// TIA Portal project "Production_Line" (V16)

(* hardware
DEVICE "S7-1200 station_1"  S7-1200 Station
   slot 0: "Rack_0"  S7-1200 Rack  Rack  V1.0
   slot 1: "PLC_1_Storage"  CPU 1214C AC/DC/Rly  6ES7 214-1BG31-0XB0  V3.0
DEVICE "S7-1200 station_2"  S7-1200 Station
   slot 0: "Rack_0"  S7-1200 Rack  Rack  V1.0
   slot 1: "PLC_3_Distribution"  CPU 1214C AC/DC/Rly  6ES7 214-1BG31-0XB0  V3.0
DEVICE "S7-1200 station_3"  S7-1200 Station
   slot 0: "Rack_0"  S7-1200 Rack  Rack  V1.0
   slot 1: "PLC_4_Measuring"  CPU 1214C AC/DC/Rly  6ES7 214-1BG31-0XB0  V3.0
DEVICE "S7-1200 station_4"  S7-1200 Station
   slot 0: "Rack_0"  S7-1200 Rack  Rack  V1.0
   slot 1: "PLC_2_P&P"  CPU 1214C AC/DC/Rly  6ES7 214-1BG31-0XB0  V3.0
DEVICE "S7-1200 station_5"  S7-1200 Station
   slot 0: "Rack_0"  S7-1200 Rack  Rack  V1.0
   slot 1: "PLC_5_Sorting"  CPU 1214C AC/DC/Rly  6ES7 214-1BG31-0XB0  V3.0
DEVICE "HMI4_Measuring"  KTP600 Basic color PN
   slot 0: "HMI4_Measuring"  KTP600 Basic color PN  6AV6 647-0AD11-3AX0  12.0.0.0
   slot 1: "HMI_RT_1"  KTP600 Basic color PN  6AV6 647-0AD11-3AX0  12.0.0.0
   slot 5: "HMI4_Measuring.IE_CP_1"  PROFINET Interface  12.0.0.0
      slot 1: "PROFINET Interface_1"  PROFINET Interface
         slot 1: "Port_1"  Port
DEVICE "HMI1_Storage"  KTP600 Basic color PN
   slot 0: "HMI1_Storage"  KTP600 Basic color PN  6AV6 647-0AD11-3AX0  12.0.0.0
   slot 1: "HMI_RT_2"  KTP600 Basic color PN  6AV6 647-0AD11-3AX0  12.0.0.0
   slot 5: "HMI1_Storage.IE_CP_1"  PROFINET Interface  12.0.0.0
      slot 1: "PROFINET Interface_1"  PROFINET Interface
         slot 1: "Port_1"  Port
*)

// ===== PLC "PLC_1_Storage"  CPU 1214C AC/DC/Rly =====

VAR_GLOBAL   // PLC tag table "Default tag table"
   "Station_homed" AT %I0.0 : Bool;
   "Error" AT %I0.1 : Bool;
   "Busy" AT %I0.2 : Bool;
   "Full" AT %I0.3 : Bool;
   "wp_at_pick" AT %I0.5 : Bool;
   "wp_not_black" AT %I0.6 : Bool;
   "wp_metallic" AT %I0.7 : Bool;
   "Home_station" AT %Q0.0 : Bool;
   "Reset_error" AT %Q0.1 : Bool;
   "Mode" AT %Q0.2 : Bool;
   "bit_0" AT %Q0.3 : Bool;
   "bit_1" AT %Q0.4 : Bool;
   "bit_2" AT %Q0.5 : Bool;
   "Strobe" AT %Q0.6 : Bool;
   "wildcard" AT %Q0.7 : Bool;
   "Rack" AT %MW1 : Int;
   "Color" AT %MW4 : Int;
   "ok" AT %M6.0 : Bool;
END_VAR

// folder: System blocks/Program resources

DATA_BLOCK "IEC_Timer_0_DB"   // DB1
{ S7_Optimized_Access := 'TRUE' }
AUTHOR : Simatic
FAMILY : IEC
NAME : IEC_TMR
VERSION : 1.0
// stored: InstanceOfName IEC_TIMER
"IEC_TIMER"
BEGIN
END_DATA_BLOCK

// folder: (top level)

FUNCTION "Select_color" : Void   // FC1, SCL
{ S7_Optimized_Access := 'TRUE' }
VERSION : 0.1
   VAR_INPUT
      color : Int;
   END_VAR
   VAR_OUTPUT
      bit0 : Bool;
      bit1 : Bool;
      bit2 : Bool;
   END_VAR
BEGIN
   CASE #color OF
       0:// red
           #bit0 := FALSE;
           #bit1 := FALSE;
           #bit2 := FALSE;
       1:// black
           #bit0 := TRUE;
           #bit1 := FALSE;
           #bit2 := FALSE;

       2:  // metallic
           #bit0 := FALSE;
           #bit1 := TRUE;
           #bit2 := FALSE;
       ELSE  // error
           #bit0 := FALSE;
           #bit1 := FALSE;
           #bit2 := FALSE;
   END_CASE;
END_FUNCTION

FUNCTION "Select_rack" : Void   // FC2, SCL
{ S7_Optimized_Access := 'TRUE' }
VERSION : 0.1
   VAR_INPUT
      Rack : Int;
   END_VAR
   VAR_OUTPUT
      bit0 : Bool;
      bit1 : Bool;
      bit2 : Bool;
   END_VAR
BEGIN
   CASE #Rack OF

       1:
           #bit0 := FALSE;
           #bit1 := FALSE;
           #bit2 := FALSE;

       2:
           #bit0 := TRUE;
           #bit1 := FALSE;
           #bit2 := FALSE;
       3:
           #bit0 := FALSE;
           #bit1 := TRUE;
           #bit2 := FALSE;

       4:
           #bit0 := TRUE;
           #bit1 := TRUE;
           #bit2 := FALSE;
       5:
           #bit0 := FALSE;
           #bit1 := FALSE;
           #bit2 := TRUE;

       6:
           #bit0 := TRUE;
           #bit1 := FALSE;
           #bit2 := TRUE;
       ELSE  // error
           #bit0 := FALSE;
           #bit1 := FALSE;
           #bit2 := FALSE;
   END_CASE;
END_FUNCTION

ORGANIZATION_BLOCK "Main"   // OB1, LAD, ProgramCycle
TITLE = "Main Program Sweep (Cycle)"
{ S7_Optimized_Access := 'TRUE' }
VERSION : 0.1
   VAR_TEMP   // added for the SCL form of the ladder/FBD networks
      _w1 : Bool;
      _w2 : Bool;
      _w3 : Bool;
   END_VAR
BEGIN

REGION Network 1
   // Remove
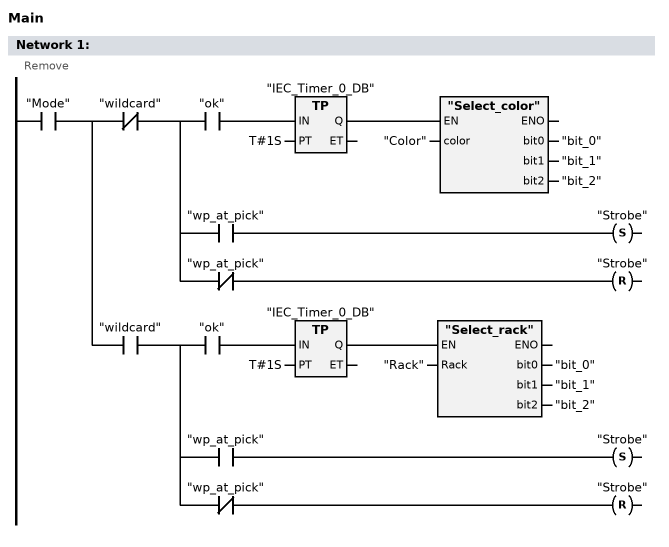
   #_w1 := "Mode" AND NOT "wildcard";
   "IEC_Timer_0_DB".TP(IN := #_w1 AND "ok", PT := T#1S);
   #_w2 := "Mode";
   IF "IEC_Timer_0_DB".Q THEN
       "Select_color"(color := "Color", bit0 => "bit_0", bit1 => "bit_1", bit2 => "bit_2");
   END_IF;
   IF #_w1 AND "wp_at_pick" THEN "Strobe" := TRUE; END_IF;
   IF #_w1 AND NOT "wp_at_pick" THEN "Strobe" := FALSE; END_IF;
   #_w3 := #_w2 AND "wildcard";
   "IEC_Timer_0_DB".TP(IN := #_w3 AND "ok", PT := T#1S);
   IF "IEC_Timer_0_DB".Q THEN
       "Select_rack"(Rack := "Rack", bit0 => "bit_0", bit1 => "bit_1", bit2 => "bit_2");
   END_IF;
   IF #_w3 AND "wp_at_pick" THEN "Strobe" := TRUE; END_IF;
   IF #_w3 AND NOT "wp_at_pick" THEN "Strobe" := FALSE; END_IF;
END_REGION
END_ORGANIZATION_BLOCK

// ===== PLC "PLC_3_Distribution"  CPU 1214C AC/DC/Rly =====

ORGANIZATION_BLOCK "Main"   // OB1, LAD, ProgramCycle
TITLE = "Main Program Sweep (Cycle)"
{ S7_Optimized_Access := 'TRUE' }
VERSION : 0.1
BEGIN
END_ORGANIZATION_BLOCK

// ===== PLC "PLC_4_Measuring"  CPU 1214C AC/DC/Rly =====

VAR_GLOBAL   // PLC tag table "Default tag table"
   "Conveyor_fwd" AT %Q0.0 : Bool;
   "Conveyor_rvs" AT %Q0.1 : Bool;
   "Adv_separator" AT %Q0.2 : Bool;
   "Retract_stopper" AT %Q0.3 : Bool;
   "Open_Gripper" AT %Q0.4 : Bool;
   "Gripper_dws" AT %Q0.5 : Bool;
   "Swivel_to_msg" AT %Q0.6 : Bool;
   "wp_beg" AT %I0.0 : Bool;
   "wp_mid" AT %I0.1 : Bool;
   "no_wp_end" AT %I0.2 : Bool;
   "Gripper_open" AT %I0.6 : Bool;
   "Gripper_raised" AT %I0.5 : Bool;
   "Swivel_at_conv" AT %I0.4 : Bool;
   "Swivel_at_msg" AT %I0.7 : Bool;
   "Analog_In" AT %IW64 : Int;
   "wp_measure" AT %MD1 : Real;
   "wp_measured" AT %M0.1 : Bool;   // Workpiece has been measured
   "shall_reject__" AT %M0.2 : Bool;
   "wp_at_conv" AT %M0.3 : Bool;
   "wp_at_msg" AT %M0.4 : Bool;
   "stopper_shall_retract" AT %M0.5 : Bool;
   "conv_shall_adv" AT %M0.6 : Bool;
   "system_ready" AT %M0.7 : Bool;
   "reset" AT %M5.0 : Bool;
END_VAR

DATA_BLOCK "Real_Main_DB"   // DB11
{ S7_Optimized_Access := 'TRUE' }
VERSION : 0.1
// stored: InstanceOfName Real_Main
"Real_Main"
BEGIN
END_DATA_BLOCK

DATA_BLOCK "General"   // DB12
{ S7_Optimized_Access := 'TRUE' }
VERSION : 0.1
   VAR
      mode_Manual : Bool;
      measured_height : Real;
      rejection_height : Real;
      operator_selected : Int;
      wp_total : Int;
      wp_ejected : Int;
      conv_direction : Bool;   // 1=forward; 0=reverse
      conv_start : Bool;   // manual
   END_VAR
BEGIN
END_DATA_BLOCK

DATA_BLOCK "Main_Manual_DB"   // DB13
{ S7_Optimized_Access := 'TRUE' }
VERSION : 0.1
// stored: InstanceOfName Main_Manual
"Main_Manual"
BEGIN
END_DATA_BLOCK

// folder: System blocks/Program resources

DATA_BLOCK "IEC_Timer_0_DB"   // DB1
{ S7_Optimized_Access := 'TRUE' }
AUTHOR : Simatic
FAMILY : IEC
NAME : IEC_TMR
VERSION : 1.0
// stored: InstanceOfName IEC_TIMER
"IEC_TIMER"
BEGIN
END_DATA_BLOCK

DATA_BLOCK "IEC_Timer_0_DB_1"   // DB2
{ S7_Optimized_Access := 'TRUE' }
AUTHOR : Simatic
FAMILY : IEC
NAME : IEC_TMR
VERSION : 1.0
// stored: InstanceOfName IEC_TIMER
"IEC_TIMER"
BEGIN
END_DATA_BLOCK

DATA_BLOCK "IEC_Timer_0_DB_2"   // DB3
{ S7_Optimized_Access := 'TRUE' }
AUTHOR : Simatic
FAMILY : IEC
NAME : IEC_TMR
VERSION : 1.0
// stored: InstanceOfName IEC_TIMER
"IEC_TIMER"
BEGIN
END_DATA_BLOCK

DATA_BLOCK "IEC_Timer_0_DB_3"   // DB4
{ S7_Optimized_Access := 'TRUE' }
AUTHOR : Simatic
FAMILY : IEC
NAME : IEC_TMR
VERSION : 1.0
// stored: InstanceOfName IEC_TIMER
"IEC_TIMER"
BEGIN
END_DATA_BLOCK

DATA_BLOCK "IEC_Timer_0_DB_4"   // DB5
{ S7_Optimized_Access := 'TRUE' }
AUTHOR : Simatic
FAMILY : IEC
NAME : IEC_TMR
VERSION : 1.0
// stored: InstanceOfName IEC_TIMER
"IEC_TIMER"
BEGIN
END_DATA_BLOCK

DATA_BLOCK "IEC_Timer_0_DB_5"   // DB6
{ S7_Optimized_Access := 'TRUE' }
AUTHOR : Simatic
FAMILY : IEC
NAME : IEC_TMR
VERSION : 1.0
// stored: InstanceOfName IEC_TIMER
"IEC_TIMER"
BEGIN
END_DATA_BLOCK

DATA_BLOCK "IEC_Timer_0_DB_6"   // DB7
{ S7_Optimized_Access := 'TRUE' }
AUTHOR : Simatic
FAMILY : IEC
NAME : IEC_TMR
VERSION : 1.0
// stored: InstanceOfName IEC_TIMER
"IEC_TIMER"
BEGIN
END_DATA_BLOCK

DATA_BLOCK "IEC_Timer_0_DB_7"   // DB8
{ S7_Optimized_Access := 'TRUE' }
AUTHOR : Simatic
FAMILY : IEC
NAME : IEC_TMR
VERSION : 1.0
// stored: InstanceOfName IEC_TIMER
"IEC_TIMER"
BEGIN
END_DATA_BLOCK

DATA_BLOCK "IEC_Timer_0_DB_8"   // DB9
{ S7_Optimized_Access := 'TRUE' }
AUTHOR : Simatic
FAMILY : IEC
NAME : IEC_TMR
VERSION : 1.0
// stored: InstanceOfName IEC_TIMER
"IEC_TIMER"
BEGIN
END_DATA_BLOCK

DATA_BLOCK "IEC_Timer_0_DB_9"   // DB10
{ S7_Optimized_Access := 'TRUE' }
AUTHOR : Simatic
FAMILY : IEC
NAME : IEC_TMR
VERSION : 1.0
// stored: InstanceOfName IEC_TIMER
"IEC_TIMER"
BEGIN
END_DATA_BLOCK

DATA_BLOCK "IEC_Counter_0_DB"   // DB14
{ S7_Optimized_Access := 'TRUE' }
AUTHOR : Simatic
FAMILY : IEC
NAME : CNTR
VERSION : 1.0
// stored: InstanceOfName IEC_COUNTER
"IEC_COUNTER"
BEGIN
END_DATA_BLOCK

DATA_BLOCK "IEC_Counter_0_DB_1"   // DB15
{ S7_Optimized_Access := 'TRUE' }
AUTHOR : Simatic
FAMILY : IEC
NAME : CNTR
VERSION : 1.0
// stored: InstanceOfName IEC_COUNTER
"IEC_COUNTER"
BEGIN
END_DATA_BLOCK

// folder: (top level)

FUNCTION_BLOCK "Real_Main"   // FB1, LAD
{ S7_Optimized_Access := 'TRUE' }
VERSION : 0.1
   VAR_TEMP   // added for the SCL form of the ladder/FBD networks
      _w1 : Bool;
   END_VAR
BEGIN

REGION Network 1: Read Measurment
   // Read Measurement
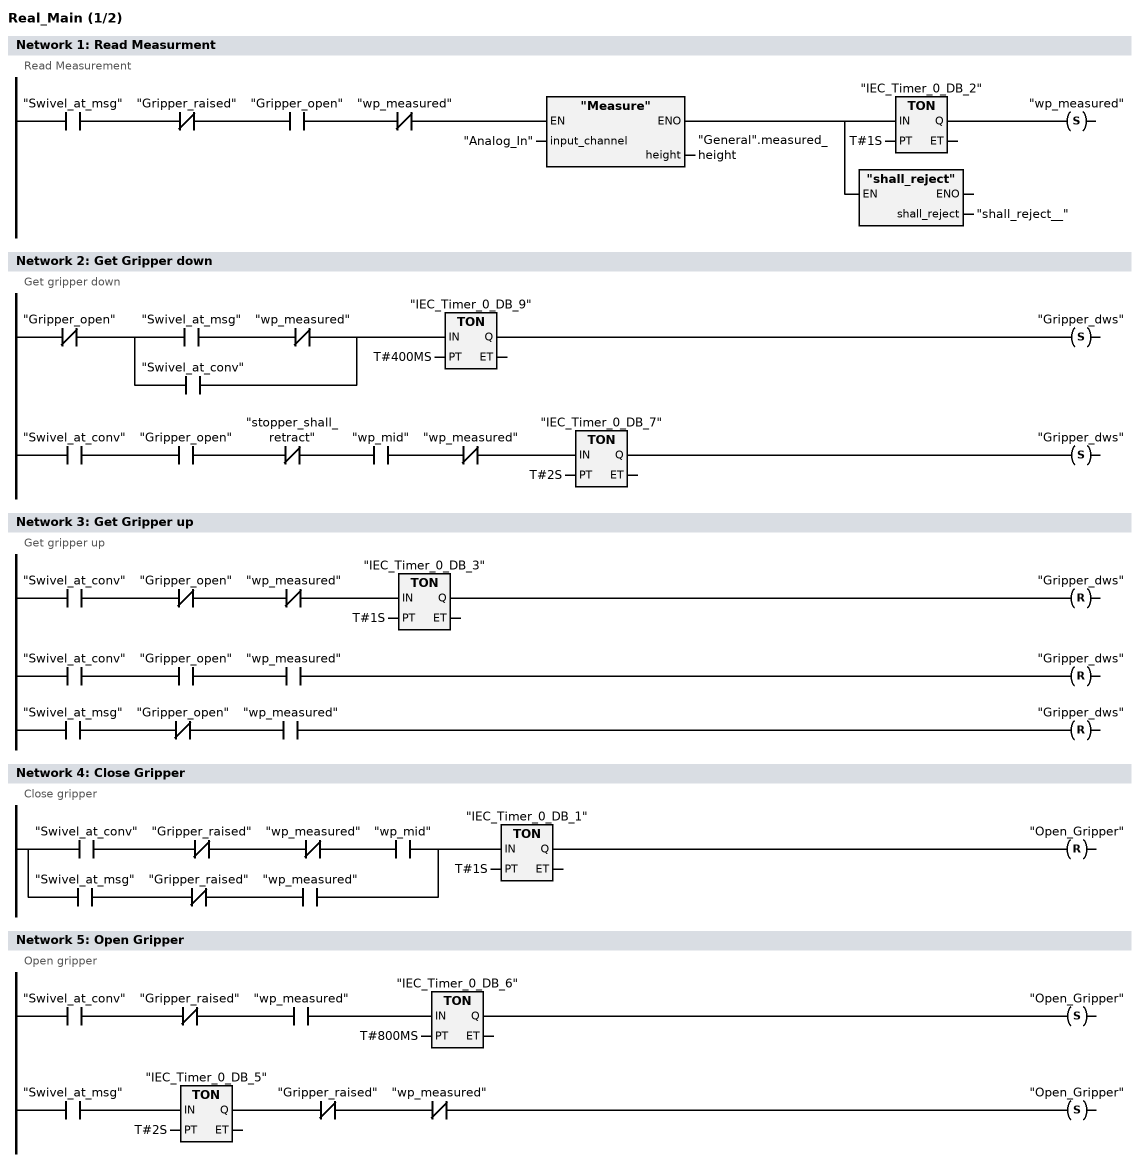
   "Measure"(EN := "Swivel_at_msg" AND NOT "Gripper_raised" AND "Gripper_open" AND NOT "wp_measured",
             input_channel := "Analog_In",
             height => "General".measured_height,
             ENO => #_w1);
   "IEC_Timer_0_DB_2".TON(IN := #_w1, PT := T#1S);
   IF "IEC_Timer_0_DB_2".Q THEN "wp_measured" := TRUE; END_IF;
   IF #_w1 THEN "shall_reject"(shall_reject => "shall_reject__"); END_IF;
END_REGION

REGION Network 2: Get Gripper down
   // Get gripper down
   "IEC_Timer_0_DB_9".TON(IN := NOT "Gripper_open" AND (("Swivel_at_msg" AND NOT "wp_measured") OR "Swivel_at_conv"),
                          PT := T#400MS);
   IF "IEC_Timer_0_DB_9".Q THEN "Gripper_dws" := TRUE; END_IF;
   "IEC_Timer_0_DB_7".TON(IN := "Swivel_at_conv" AND "Gripper_open" AND NOT "stopper_shall_retract" AND "wp_mid" AND NOT "wp_measured",
                          PT := T#2S);
   IF "IEC_Timer_0_DB_7".Q THEN "Gripper_dws" := TRUE; END_IF;
END_REGION

REGION Network 3: Get Gripper up
   // Get gripper up
   "IEC_Timer_0_DB_3".TON(IN := "Swivel_at_conv" AND NOT "Gripper_open" AND NOT "wp_measured", PT := T#1S);
   IF "IEC_Timer_0_DB_3".Q THEN "Gripper_dws" := FALSE; END_IF;
   IF "Swivel_at_conv" AND "Gripper_open" AND "wp_measured" THEN "Gripper_dws" := FALSE; END_IF;
   IF "Swivel_at_msg" AND NOT "Gripper_open" AND "wp_measured" THEN "Gripper_dws" := FALSE; END_IF;
END_REGION

REGION Network 4: Close Gripper
   // Close gripper
   "IEC_Timer_0_DB_1".TON(IN := ("Swivel_at_conv" AND NOT "Gripper_raised" AND NOT "wp_measured" AND "wp_mid") OR ("Swivel_at_msg" AND NOT "Gripper_raised" AND "wp_measured"),
                          PT := T#1S);
   IF "IEC_Timer_0_DB_1".Q THEN "Open_Gripper" := FALSE; END_IF;
END_REGION

REGION Network 5: Open Gripper
   // Open gripper
   "IEC_Timer_0_DB_6".TON(IN := "Swivel_at_conv" AND NOT "Gripper_raised" AND "wp_measured", PT := T#800MS);
   IF "IEC_Timer_0_DB_6".Q THEN "Open_Gripper" := TRUE; END_IF;
   "IEC_Timer_0_DB_5".TON(IN := "Swivel_at_msg", PT := T#2S);
   IF "IEC_Timer_0_DB_5".Q AND NOT "Gripper_raised" AND NOT "wp_measured" THEN
       "Open_Gripper" := TRUE;
   END_IF;
END_REGION

REGION Network 6: Get swivel to measuring station
   // Get swivel to measuring station
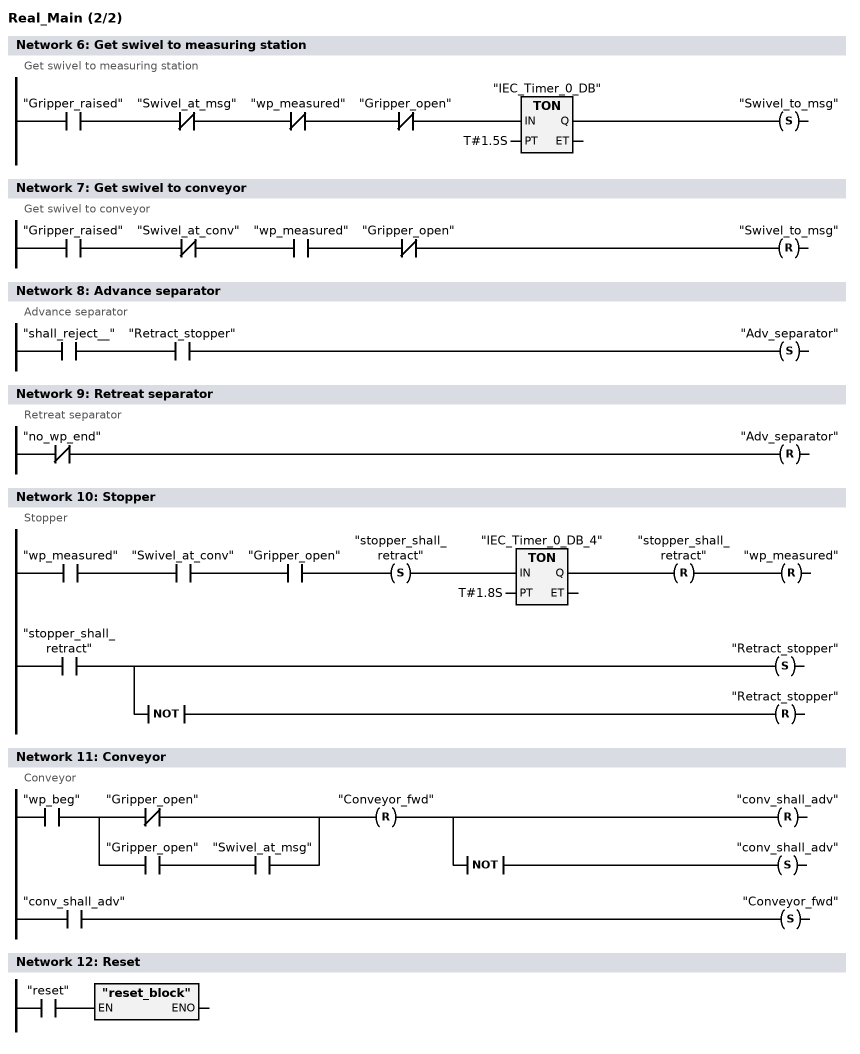
   "IEC_Timer_0_DB".TON(IN := "Gripper_raised" AND NOT "Swivel_at_msg" AND NOT "wp_measured" AND NOT "Gripper_open",
                        PT := T#1.5S);
   IF "IEC_Timer_0_DB".Q THEN "Swivel_to_msg" := TRUE; END_IF;
END_REGION

REGION Network 7: Get swivel to conveyor
   // Get swivel to conveyor
   RUNG wire#powerrail
      Contact( "Gripper_raised" )
      I_Contact( "Swivel_at_conv" )
      Contact( "wp_measured" )
      I_Contact( "Gripper_open" )
      R_Coil( "Swivel_to_msg" )
   END_RUNG
   // the same network as SCL:
   IF "Gripper_raised" AND NOT "Swivel_at_conv" AND "wp_measured" AND NOT "Gripper_open" THEN
       "Swivel_to_msg" := FALSE;
   END_IF;
END_REGION

REGION Network 8: Advance separator
   // Advance separator
   RUNG wire#powerrail
      Contact( "shall_reject__" )
      Contact( "Retract_stopper" )
      S_Coil( "Adv_separator" )
   END_RUNG
   // the same network as SCL:
   IF "shall_reject__" AND "Retract_stopper" THEN "Adv_separator" := TRUE; END_IF;
END_REGION

REGION Network 9: Retreat separator
   // Retreat separator
   RUNG wire#powerrail
      I_Contact( "no_wp_end" )
      R_Coil( "Adv_separator" )
   END_RUNG
   // the same network as SCL:
   IF NOT "no_wp_end" THEN "Adv_separator" := FALSE; END_IF;
END_REGION

REGION Network 10: Stopper
   // Stopper
   #_w1 := "wp_measured" AND "Swivel_at_conv" AND "Gripper_open";
   IF #_w1 THEN "stopper_shall_retract" := TRUE; END_IF;
   "IEC_Timer_0_DB_4".TON(IN := #_w1, PT := T#1.8S);
   IF "IEC_Timer_0_DB_4".Q THEN
       "stopper_shall_retract" := FALSE;
       "wp_measured" := FALSE;
   END_IF;
   IF "stopper_shall_retract" THEN "Retract_stopper" := TRUE; END_IF;
   IF NOT "stopper_shall_retract" THEN "Retract_stopper" := FALSE; END_IF;
END_REGION

REGION Network 11: Conveyor
   // Conveyor
   RUNG wire#powerrail
      Contact( "wp_beg" )
      wire#w1
      I_Contact( "Gripper_open" )
      wire#w2
      R_Coil( "Conveyor_fwd" )
      wire#w3
      R_Coil( "conv_shall_adv" )
   END_RUNG
   RUNG wire#w1
      Contact( "Gripper_open" )
      Contact( "Swivel_at_msg" )
   END_RUNG wire#w2
   RUNG wire#w3
      Not()
      S_Coil( "conv_shall_adv" )
   END_RUNG
   RUNG wire#powerrail
      Contact( "conv_shall_adv" )
      S_Coil( "Conveyor_fwd" )
   END_RUNG
   // the same network as SCL:
   #_w1 := "wp_beg" AND (NOT "Gripper_open" OR ("Gripper_open" AND "Swivel_at_msg"));
   IF #_w1 THEN
       "Conveyor_fwd" := FALSE;
       "conv_shall_adv" := FALSE;
   END_IF;
   IF NOT #_w1 THEN "conv_shall_adv" := TRUE; END_IF;
   IF "conv_shall_adv" THEN "Conveyor_fwd" := TRUE; END_IF;
END_REGION

REGION Network 12: Reset
   RUNG wire#powerrail
      Contact( "reset" )
      "reset_block"()
   END_RUNG
   // the same network as SCL:
   IF "reset" THEN "reset_block"(); END_IF;
END_REGION
END_FUNCTION_BLOCK

FUNCTION_BLOCK "Main_Manual"   // FB2, LAD
{ S7_Optimized_Access := 'TRUE' }
VERSION : 0.1
BEGIN

REGION Network 1
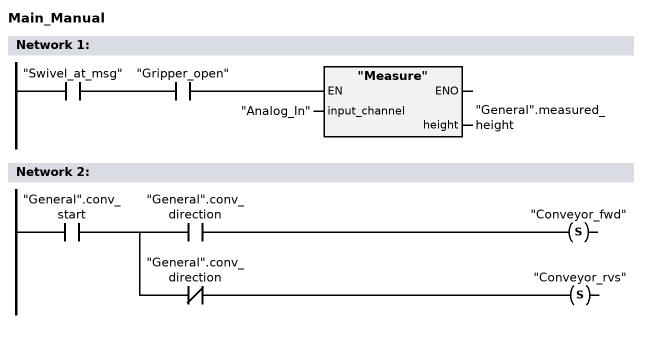
   RUNG wire#powerrail
      Contact( "Swivel_at_msg" )
      Contact( "Gripper_open" )
      "Measure"(input_channel := "Analog_In", height => "General".measured_height)
   END_RUNG
   // the same network as SCL:
   IF "Swivel_at_msg" AND "Gripper_open" THEN
       "Measure"(input_channel := "Analog_In", height => "General".measured_height);
   END_IF;
END_REGION

REGION Network 2
   RUNG wire#powerrail
      Contact( "General".conv_start )
      wire#w1
      Contact( "General".conv_direction )
      S_Coil( "Conveyor_fwd" )
   END_RUNG
   RUNG wire#w1
      I_Contact( "General".conv_direction )
      S_Coil( "Conveyor_rvs" )
   END_RUNG
   // the same network as SCL:
   IF "General".conv_start AND "General".conv_direction THEN "Conveyor_fwd" := TRUE; END_IF;
   IF "General".conv_start AND NOT "General".conv_direction THEN "Conveyor_rvs" := TRUE; END_IF;
END_REGION
END_FUNCTION_BLOCK

FUNCTION "reset_block" : Void   // FC1, LAD
{ S7_Optimized_Access := 'TRUE' }
VERSION : 0.1
BEGIN

REGION Network 1
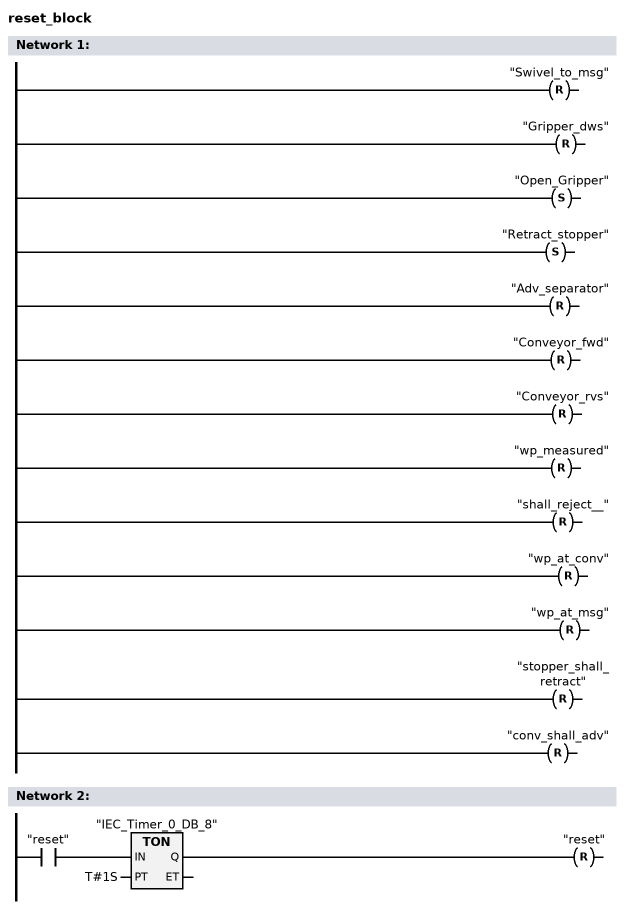
   RUNG wire#powerrail
      R_Coil( "Swivel_to_msg" )
   END_RUNG
   RUNG wire#powerrail
      R_Coil( "Gripper_dws" )
   END_RUNG
   RUNG wire#powerrail
      S_Coil( "Open_Gripper" )
   END_RUNG
   RUNG wire#powerrail
      S_Coil( "Retract_stopper" )
   END_RUNG
   RUNG wire#powerrail
      R_Coil( "Adv_separator" )
   END_RUNG
   RUNG wire#powerrail
      R_Coil( "Conveyor_fwd" )
   END_RUNG
   RUNG wire#powerrail
      R_Coil( "Conveyor_rvs" )
   END_RUNG
   RUNG wire#powerrail
      R_Coil( "wp_measured" )
   END_RUNG
   RUNG wire#powerrail
      R_Coil( "shall_reject__" )
   END_RUNG
   RUNG wire#powerrail
      R_Coil( "wp_at_conv" )
   END_RUNG
   RUNG wire#powerrail
      R_Coil( "wp_at_msg" )
   END_RUNG
   RUNG wire#powerrail
      R_Coil( "stopper_shall_retract" )
   END_RUNG
   RUNG wire#powerrail
      R_Coil( "conv_shall_adv" )
   END_RUNG
   // the same network as SCL:
   "Swivel_to_msg" := FALSE;
   "Gripper_dws" := FALSE;
   "Open_Gripper" := TRUE;
   "Retract_stopper" := TRUE;
   "Adv_separator" := FALSE;
   "Conveyor_fwd" := FALSE;
   "Conveyor_rvs" := FALSE;
   "wp_measured" := FALSE;
   "shall_reject__" := FALSE;
   "wp_at_conv" := FALSE;
   "wp_at_msg" := FALSE;
   "stopper_shall_retract" := FALSE;
   "conv_shall_adv" := FALSE;
END_REGION

REGION Network 2
   "IEC_Timer_0_DB_8".TON(IN := "reset", PT := T#1S);
   IF "IEC_Timer_0_DB_8".Q THEN "reset" := FALSE; END_IF;
END_REGION
END_FUNCTION

FUNCTION "shall_reject" : Void   // FC2, SCL
{ S7_Optimized_Access := 'TRUE' }
VERSION : 0.1
   VAR_OUTPUT
      shall_reject : Bool;
   END_VAR
BEGIN
   CASE "General".operator_selected OF
       0: //greater than
           IF "General".measured_height > "General".rejection_height THEN
               #shall_reject := TRUE;
           ELSE
               #shall_reject := FALSE;
           END_IF;
           ;
       1: //less than
           IF "General".measured_height < "General".rejection_height THEN
               #shall_reject := TRUE;
           ELSE
               #shall_reject := FALSE;
           END_IF;
           ;
       2: // greater or equal than
           IF "General".measured_height >= "General".rejection_height THEN
               #shall_reject := TRUE;
           ELSE
               #shall_reject := FALSE;
           END_IF;
           ;
       3: // less or equal than
           IF "General".measured_height <= "General".rejection_height THEN
               #shall_reject := TRUE;
           ELSE
               #shall_reject := FALSE;
           END_IF;
           ;

   END_CASE;
END_FUNCTION

FUNCTION "Measure" : Void   // FC4, LAD
{ S7_Optimized_Access := 'TRUE' }
VERSION : 0.1
   VAR_INPUT
      input_channel : Int;
   END_VAR
   VAR_OUTPUT
      height : Real;
   END_VAR
   VAR_TEMP
      temp1 : Real;
      measuring : Real;
   END_VAR
   VAR CONSTANT
      cap_det : Real := 25.5;
      max_distance : Real := 74.0;
      min_distance : Real := 46.0;
   END_VAR
BEGIN

REGION Network 1
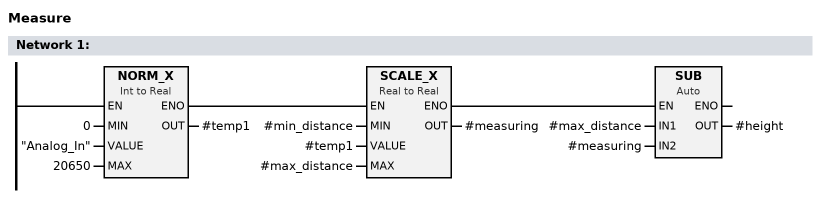
   RUNG wire#powerrail
      { S7_Templates := "[SrcType := Int, DestType := Real]"; S7_GenerateENO := "TRUE" } Normalize(min := 0, value := "Analog_In", max := 20650, out => #temp1)
      { S7_Templates := "[SrcType := Real, DestType := Real]"; S7_GenerateENO := "TRUE" } Scale(min := #min_distance, value := #temp1, max := #max_distance, out => #measuring)
      { S7_GenerateENO := "TRUE" } Sub(in1 := #max_distance, in2 := #measuring, out => #height)
   END_RUNG
   // the same network as SCL:
   // ENO of a box is taken as its EN; it also drops when the box reports an error
   #temp1 := NORM_X(MIN := 0, VALUE := "Analog_In", MAX := 20650);
   #measuring := SCALE_X(MIN := #min_distance, VALUE := #temp1, MAX := #max_distance);
   #height := #max_distance - #measuring;
END_REGION
END_FUNCTION

ORGANIZATION_BLOCK "Main"   // OB1, LAD, ProgramCycle
TITLE = "Main Program Sweep (Cycle)"
{ S7_Optimized_Access := 'TRUE' }
VERSION : 0.1
   VAR_TEMP   // added for the SCL form of the ladder/FBD networks
      _w1 : Bool;
      _w2 : Bool;
   END_VAR
BEGIN

REGION Network 1
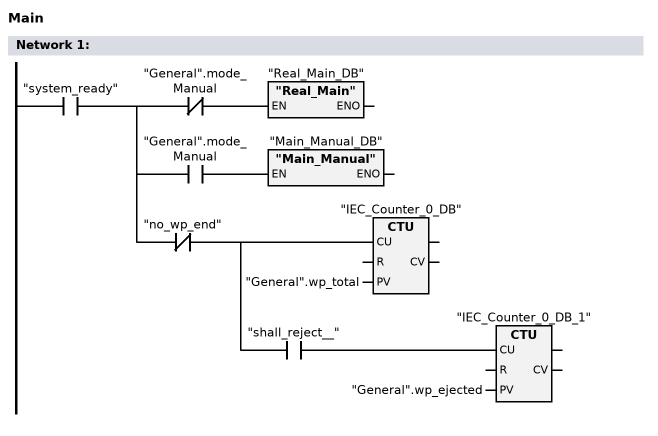
   #_w1 := "system_ready";
   IF "system_ready" AND NOT "General".mode_Manual THEN
       "Real_Main_DB"();   // "Real_Main"
   END_IF;
   IF #_w1 AND "General".mode_Manual THEN
       "Main_Manual_DB"();   // "Main_Manual"
   END_IF;
   #_w2 := #_w1 AND NOT "no_wp_end";
   "IEC_Counter_0_DB".CTU(CU := #_w2, PV := "General".wp_total);
   "IEC_Counter_0_DB_1".CTU(CU := #_w2 AND "shall_reject__", PV := "General".wp_ejected);
END_REGION
END_ORGANIZATION_BLOCK

ORGANIZATION_BLOCK "Startup"   // OB100, LAD, Startup
TITLE = "Complete Restart"
{ S7_Optimized_Access := 'TRUE' }
VERSION : 0.1
   VAR_INPUT
      LostRetentive : Bool;   // True if retentive data are lost
      LostRTC : Bool;   // True if date and time are lost
   END_VAR
BEGIN

REGION Network 1
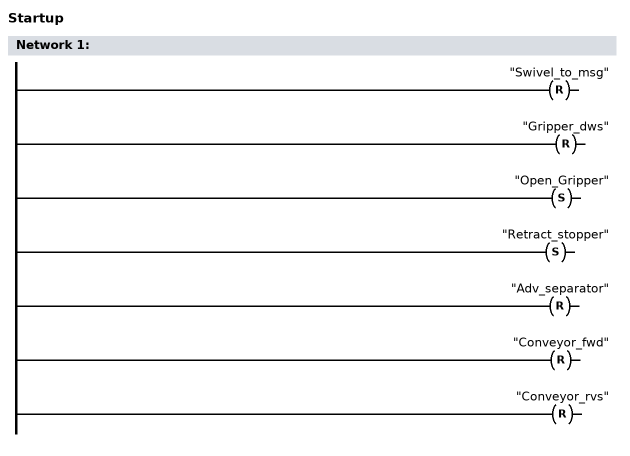
   RUNG wire#powerrail
      R_Coil( "Swivel_to_msg" )
   END_RUNG
   RUNG wire#powerrail
      R_Coil( "Gripper_dws" )
   END_RUNG
   RUNG wire#powerrail
      S_Coil( "Open_Gripper" )
   END_RUNG
   RUNG wire#powerrail
      S_Coil( "Retract_stopper" )
   END_RUNG
   RUNG wire#powerrail
      R_Coil( "Adv_separator" )
   END_RUNG
   RUNG wire#powerrail
      R_Coil( "Conveyor_fwd" )
   END_RUNG
   RUNG wire#powerrail
      R_Coil( "Conveyor_rvs" )
   END_RUNG
   // the same network as SCL:
   "Swivel_to_msg" := FALSE;
   "Gripper_dws" := FALSE;
   "Open_Gripper" := TRUE;
   "Retract_stopper" := TRUE;
   "Adv_separator" := FALSE;
   "Conveyor_fwd" := FALSE;
   "Conveyor_rvs" := FALSE;
END_REGION
END_ORGANIZATION_BLOCK

// ===== PLC "PLC_2_P&P"  CPU 1214C AC/DC/Rly =====

ORGANIZATION_BLOCK "Main"   // OB1, LAD, ProgramCycle
TITLE = "Main Program Sweep (Cycle)"
{ S7_Optimized_Access := 'TRUE' }
VERSION : 0.1
BEGIN
END_ORGANIZATION_BLOCK

// ===== PLC "PLC_5_Sorting"  CPU 1214C AC/DC/Rly =====

ORGANIZATION_BLOCK "Main"   // OB1, LAD, ProgramCycle
TITLE = "Main Program Sweep (Cycle)"
{ S7_Optimized_Access := 'TRUE' }
VERSION : 0.1
BEGIN
END_ORGANIZATION_BLOCK

(* ===== HMI "HMI_RT_1" =====
system functions are stored by id; their names below are inferred from use
connection "HMI_Connection_1": ETHERNET, SMART_S7_1200_OMS

HMI tags "Default tag table"
   "Tag_ScreenNumber" : UInt, internal
   "wp_beg" : Bool = PLC wp_beg AT %I0.0, 1 s
   "wp_mid" : Bool = PLC wp_mid AT %I0.1, 1 s
   "no_wp_end" : Bool = PLC no_wp_end AT %I0.2, 1 s
   "reset" : Bool = PLC reset AT %M5.0, 1 s
   "system_ready" : Bool = PLC system_ready AT %M0.7, 1 s
   "Gripper_open" : Bool = PLC Gripper_open AT %I0.6, 1 s
   "Swivel_at_conv" : Bool = PLC Swivel_at_conv AT %I0.4, 1 s
   "Swivel_at_msg" : Bool = PLC Swivel_at_msg AT %I0.7, 1 s
   "Gripper_raised" : Bool = PLC Gripper_raised AT %I0.5, 1 s
   "General_rejection_height" : Real = PLC General.rejection_height, 1 s
   "General_operator_selected" : Int = PLC General.operator_selected, 1 s
   "Adv_separator" : Bool = PLC Adv_separator AT %Q0.2, 1 s
   "Retract_stopper" : Bool = PLC Retract_stopper AT %Q0.3, 1 s
   "Swivel_to_msg" : Bool = PLC Swivel_to_msg AT %Q0.6, 1 s
   "Open_Gripper" : Bool = PLC Open_Gripper AT %Q0.4, 1 s
   "Gripper_dws" : Bool = PLC Gripper_dws AT %Q0.5, 1 s
   "General_measured_height" : Real = PLC General.measured_height, 1 s
   "General_wp_ejected" : Int = PLC General.wp_ejected, 1 s
   "General_wp_total" : Int = PLC General.wp_total, 1 s
   "General_conv_direction" : Bool = PLC General.conv_direction, 1 s
   "General_conv_start" : Bool = PLC General.conv_start, 1 s
   "Conveyor_fwd" : Bool = PLC Conveyor_fwd AT %Q0.0, 1 s
   "Conveyor_rvs" : Bool = PLC Conveyor_rvs AT %Q0.1, 1 s

text list "height_operators": 0 '<'; 1 '<='; 2 '>'; 3 '>='

text list "Gripper_altitude": 0 'DOWN'; 1 'UP'

text list "Gripper": 0 'CLOSED'; 1 'OPEN'

graphic list "Operators": 0 'greater_than_1'; 1 'less_than'; 2 'greaterORequal_than'; 3 'lessORequal_than'; 4 'Press here'

screen "Inventory" 320x240, template "Template_1"
   on GenerateScreen: SetTag("Tag_ScreenNumber", 5)
   TextField "Text field_1" at 97,0 size 121x31; Text 'Inventory'
   TextField "Text field_2" at 17,70 size 61x21; Text 'On Rail'
   TextField "Text field_3" at 126,103 size 132x21; Text 'Total Processed'
   IOField "I/O field_2" at 272,103 size 39x26; FormatPattern 99
      ProcessValue <- "General_wp_total"
   Bar "Bar_1" at 4,103 size 96x76; MinimumValue 0; MaximumValue 6
      ProcessValue <- "General_wp_ejected"
   Button "Button_1" at 121,158 size 65x22; TextOff 'Clear Rail'
      on Press: SetTag("General_wp_ejected", 0)
   Button "Button_2" at 206,158 size 96x22; TextOff 'Clear Processed'
      on Press: SetTag("General_wp_total", 0)

Template "Template_1" 320x240
   Button "Exit" at 266,202 size 52x37; TextOff 'Exit'; PictureOff "ExitRuntime_KTP600_Basic_color_PN"; PictureOn "ExitRuntime_KTP600_Basic_color_PN"
      on Release: StopRuntime(0)
   Button "Template_Button_1" at 160,202 size 52x37; TextOff 'RESET'
      on Press: SetBit("reset")
   Button "Template_Button_2" at 107,202 size 52x37; TextOff 'STOP'; PictureOff "stop"; PictureOn "start"
      on Press: ResetBit("system_ready")
   Button "Start screen" at 1,202 size 52x37; TextOff 'Start screen'; PictureOff "NavigateHome_KTP600_Basic_color_PN"; PictureOn "NavigateHome_KTP600_Basic_color_PN"
      on Release: ActivateScreen("Home", 0)
   DateTimeField "HmiScreenItemData" at 235,19 size 85x19
   DateTimeField "HmiScreenItemData_1" at 235,0 size 85x19
   GraphicView "Logo" at 0,0 size 54x50; Picture "Unisabana"

screen "Home" 320x240, template "Template_1"
   on GenerateScreen: SetTag("Tag_ScreenNumber", 1)
   Button "Set up" at 198,121 size 104x30; TextOff 'Set up'
      on Release: ActivateScreen("Set up", 0)
   Button "Start" at 198,46 size 104x30; TextOff 'Start'
      on Release: ActivateScreen("Start", 0)
      on Press: SetBit("system_ready")
   Button "Manual" at 198,162 size 104x30; TextOff 'Manual'; Authorization "Manual"
      on Release: ActivateScreen("Manual", 0)
   Button "Inventory" at 198,81 size 104x30; TextOff 'Inventory'
      on Release: ActivateScreen("Inventory", 0)
   GraphicView "Graphic view_1" at 20,46 size 146x130; Picture "measuring_noBackground"
   TextField "Text field_1" at 63,4 size 176x25; Text 'Measuring Station'

screen "Set up" 320x240, template "Template_1"
   on GenerateScreen: SetTag("Tag_ScreenNumber", 2)
   TextField "Text field_1" at 112,5 size 81x31; Text 'Set Up'
   TextField "Text field_2" at 9,76 size 139x21; Text 'Rejection Height'
   TextField "Text field_4" at 273,76 size 24x18; Text 'mm'
   IOField "I/O field_1" at 219,76 size 50x23; FormatPattern s999999999.999
      ProcessValue <- "General_rejection_height"
   GraphicIOField "Graphic I/O field_1" at 172,66 size 42x41; PictureList "Operators"
      ProcessValue <- "General_operator_selected"

screen "Start" 320x240, template "More_Space"
   on GenerateScreen: SetTag("Tag_ScreenNumber", 3)
   GraphicView "Graphic view_1" at 29,192 size 243x48; Picture "conveyor_1"
   Circle "Circle_1" at 69,174 size 22x22
      Visibility <- "wp_beg"
   Circle "Circle_2" at 139,174 size 22x22
      Visibility <- "wp_mid"
   Circle "Circle_3" at 222,174 size 22x22
      Visibility <- "no_wp_end"
   IOField "I/O field_1" at 148,30 size 67x23; FormatPattern 99.99; Unit  mm
      ProcessValue <- "General_measured_height"
   TextField "Text field_6" at 60,35 size 82x18; Text 'Piece Height'
   TextField "Text field_1" at 173,81 size 63x21; Text 'Gripper'
   SymbolicIOField "Symbolic I/O field_1" at 173,132 size 55x17; TextOff '0'; TextOn '1'; TextList "Gripper"
      ProcessValue <- "Gripper_open"
   TextField "Text field_2" at 8,109 size 55x18; Text 'Conveyor'
   Circle "Circle_4" at 77,108 size 19x19
      Appearance <- "Swivel_at_conv"
   TextField "Text field_3" at 8,133 size 61x18; Text 'Measuring'
   Circle "Circle_5" at 77,132 size 19x19
      Appearance <- "Swivel_at_msg"
   SymbolicIOField "Symbolic I/O field_2" at 173,109 size 55x17; TextOff '0'; TextOn '1'; TextList "Gripper_altitude"
      ProcessValue <- "Gripper_raised"
   TextField "Text field_4" at 19,78 size 77x21; Text 'Swivel at'

screen "Manual" 320x240, template "More_Space"
   on GenerateScreen: SetTag("Tag_ScreenNumber", 4); function_f23ef4c9(); SetBit("reset"); SetBit("system_ready")
   GraphicView "Graphic view_1" at 17,88 size 233x47; Picture "conveyor_1"
   TextField "Text field_1" at 9,133 size 64x18; Text 'Conveyor'
   Switch "Switch_1" at 9,155 size 64x32; CaptionText 'Switch'; TextOff 'Reverse'; TextOn 'Forward'
      ProcessValue <- "General_conv_direction"
   Switch "Switch_2" at 14,191 size 49x41; CaptionText 'Switch'; TextOff 'OFF'; TextOn 'ON'; PictureOn "stop"; PictureOff "start"
      ProcessValue <- "General_conv_start"
      on SwitchOff: ResetBit("Conveyor_fwd"); ResetBit("Conveyor_rvs")
   TextField "Text field_2" at 250,129 size 68x18; Text 'Separator'
   Switch "Switch_3" at 250,147 size 64x32; TextOn 'ON'; CaptionText 'Switch'; TextOff 'OFF'
      ProcessValue <- "Adv_separator"
   TextField "Text field_3" at 250,182 size 54x18; Text 'Stopper'
   Switch "Switch_4" at 250,200 size 64x32; TextOn 'Retracted'; CaptionText 'Switch'; TextOff 'Released'
      ProcessValue <- "Retract_stopper"
   TextField "Text field_5" at 103,169 size 49x18; Text 'Gripper'
   Switch "Switch_6" at 158,191 size 46x35; TextOn 'Open'; CaptionText 'Switch'; TextOff 'Close'
      ProcessValue <- "Open_Gripper"
   Switch "Switch_7" at 106,191 size 46x35; TextOn 'Down'; CaptionText 'Switch'; TextOff 'Up'
      ProcessValue <- "Gripper_dws"
   TextField "Text field_4" at 250,79 size 43x18; Text 'Swivel'
   Switch "Switch_5" at 250,97 size 64x32; TextOn 'Measure'; CaptionText 'Switch'; TextOff 'Conveyor'
      ProcessValue <- "Swivel_to_msg"
   Circle "Circle_1" at 40,69 size 22x22
      Visibility <- "wp_beg"
   Circle "Circle_2" at 110,69 size 22x22
      Visibility <- "wp_mid"
   Circle "Circle_3" at 193,69 size 22x22
      Visibility <- "no_wp_end"
   IOField "I/O field_1" at 152,15 size 67x23; FormatPattern 99.99; Unit  mm
      ProcessValue <- "General_measured_height"
   TextField "Text field_6" at 63,15 size 82x18; Text 'Piece Height'

Template "More_Space" 320x240
   Button "Template_Button_1" at 266,40 size 52x37; TextOff 'RESET'
      on Press: SetBit("reset")
   Button "Template_Button_2" at 266,0 size 52x37; TextOff 'STOP'; PictureOn "start"; PictureOff "stop"
      on Press: ResetBit("system_ready")
   Button "Start screen" at 0,0 size 52x37; TextOn 'Start screen'; TextOff 'Start screen'; PictureOn "NavigateHome_KTP600_Basic_color_PN"; PictureOff "NavigateHome_KTP600_Basic_color_PN"
      on Release: ActivateScreen("Home", 0)
*)

(* ===== HMI "HMI_RT_2" =====
system functions are stored by id; their names below are inferred from use
connection "HMI_Connection_2": ETHERNET, SMART_S7_1200_OMS

HMI tags "Default tag table"
   "Color" : Int = PLC Color AT %MW4, 1 s
   "color_hmi" : Int, internal
   "Mode" : Bool = PLC Mode AT %Q0.2, 1 s
   "ok" : Bool = PLC ok AT %M6.0, 1 s
   "Rack" : Int = PLC Rack AT %MW1, 1 s
   "rack_hmi" : Int AT %DB1.DBX0.0
   "Tag_ScreenNumber" : UInt, internal
   "wildcard" : Bool = PLC wildcard AT %Q0.7, 1 s

text list "Colors": 0 'Red'; 1 'Black'; 2 'Metallic'

text list "Racks": 1 'Rack 1'; 2 'Rack 2'; 3 'Rack 3'; 4 'Rack 4'; 5 'Rack 5'; 6 'Rack 6'

Template "Template_1" 320x240
   Button "Exit" at 266,202 size 52x37; TextOff 'Exit'; PictureOff "ExitRuntime_KTP600_Basic_color_PN"; PictureOn "ExitRuntime_KTP600_Basic_color_PN"
      on Release: StopRuntime(0)
   Button "Start screen" at 1,202 size 52x37; TextOff 'Start screen'; PictureOff "NavigateHome_KTP600_Basic_color_PN"; PictureOn "NavigateHome_KTP600_Basic_color_PN"
      on Release: ActivateScreen("Root screen", 0)
   DateTimeField "HmiScreenItemData" at 235,19 size 85x19
   DateTimeField "HmiScreenItemData_1" at 235,0 size 85x19
   GraphicView "Logo" at 0,0 size 38x38; Picture "Logo of HMI_1"

screen "Color" 320x240, template "Template_1"
   on GenerateScreen: SetTag("Tag_ScreenNumber", 6)
   Button "Back" at 1,39 size 41x35; TextOn 'Back'; TextOff 'Back'; PictureOff "Left_Arrow"
      on Release: ActivateScreen("Remove", 0)
   SymbolicIOField "Symbolic I/O field_1" at 32,126 size 96x17; TextOn '1'; TextOff '0'; TextList "Colors"
      ProcessValue <- "color_hmi"
   Button "Button_1" at 192,121 size 96x32; TextOff 'OK'
      on Release: ResetBit("ok")
      on Press: SetTag("Color", "color_hmi"); SetBit("ok")
   TextField "Text field_1" at 32,97 size 52x21; Text 'Select'

screen "Manual" 320x240, template "Template_1"
   on GenerateScreen: SetTag("Tag_ScreenNumber", 3)
   Button "Back" at 1,39 size 39x32; TextOn 'Back'; TextOff 'Back'; PictureOff "Left_Arrow"
      on Release: ActivateScreen("Place", 0)
   SymbolicIOField "Symbolic I/O field_1" at 20,130 size 96x17; TextOn '1'; TextOff '0'; TextList "Racks"
      ProcessValue <- "rack_hmi"
   Button "Button_1" at 201,126 size 96x32; TextOff 'OK'
      on Press: SetTag("Rack", "rack_hmi")
   TextField "Text field_1" at 19,102 size 52x21; Text 'Select'

screen "Place" 320x240, template "Template_1"
   on GenerateScreen: SetTag("Tag_ScreenNumber", 2)
   Button "Back" at 1,39 size 40x35; TextOn 'Back'; TextOff 'Back'; PictureOff "Left_Arrow"
      on Release: ActivateScreen("Root screen", 0)
   Button "Manual" at 177,120 size 104x30; TextOn 'Manual'; TextOff 'Manual'
      on Release: ActivateScreen("Manual", 0)
      on Press: SetBit("wildcard")
   Button "Button_1" at 51,120 size 103x30; TextOff 'Auto'
      on Press: ResetBit("wildcard")

screen "Racks" 320x240, template "Template_1"
   on GenerateScreen: SetTag("Tag_ScreenNumber", 5)
   Button "Back" at 1,39 size 39x32; TextOn 'Back'; TextOff 'Back'; PictureOff "Left_Arrow"
      on Release: ActivateScreen("Remove", 0)
   SymbolicIOField "Symbolic I/O field_1" at 36,126 size 96x17; TextOn '1'; TextOff '0'; TextList "Racks"
      ProcessValue <- "rack_hmi"
   Button "Button_1" at 198,124 size 96x32; TextOff 'OK'
      on Release: ResetBit("ok")
      on Press: SetTag("Rack", "rack_hmi"); SetBit("ok")
   TextField "Text field_1" at 36,100 size 52x21; Text 'Select'

screen "Remove" 320x240, template "Template_1"
   on GenerateScreen: SetTag("Tag_ScreenNumber", 4)
   Button "Back" at 1,39 size 40x36; TextOn 'Back'; TextOff 'Back'; PictureOff "Left_Arrow"
      on Release: ActivateScreen("Root screen", 0)
   Button "Racks" at 41,118 size 104x30; TextOn 'Racks'; TextOff 'Racks'
      on Release: ActivateScreen("Racks", 0)
      on Press: SetBit("wildcard")
   Button "Color" at 166,118 size 104x30; TextOn 'Color'; TextOff 'Color'
      on Release: ActivateScreen("Color", 0)
      on Press: ResetBit("wildcard")

screen "Root screen" 320x240, template "Template_1"
   on GenerateScreen: SetTag("Tag_ScreenNumber", 1)
   Button "Place" at 197,81 size 104x30; TextOn 'Place'; TextOff 'Place'
      on Release: ActivateScreen("Place", 0)
      on Press: ResetBit("Mode")
   Button "Remove" at 197,134 size 104x30; TextOn 'Remove'; TextOff 'Remove'
      on Release: ActivateScreen("Remove", 0)
      on Press: SetBit("Mode")
   GraphicView "Graphic view_1" at 41,44 size 135x152; Picture "storage"
   TextField "Text field_1" at 88,1 size 95x31; Text 'Storage'
*)